(* CODESYS project UralKoksWin.project

Project tree, tasks and I/O mapping:
  Device : SPK1xx[M01], Production association OWEN, order no. 4, version 3.5.11.54
    application Application
      libraries: Standard, * (System); Util, * (System)
      task MainTask (cyclic, interval t#20ms, priority 1) calls PLC_PRG, MECH
      task VISU_TASK (cyclic, interval 100 ms, priority 31) calls VisuElems.Visu_Prg, CountWebCli
      task Task_Chain (cyclic, interval t#20ms, priority 1) calls Chain
      task TrendRecordingTask (cyclic, interval 100 ms, priority 31) calls VisuTrendStorageAccess.GlobalInstances.g_TrendRecordingManager.CyclicCall
      program PLC_PRG [LD]
      visualisation VFrADiag
      data type MV210_202
      data type MU210_402
      data type Vector75
      visualisation VMain
      visualisation VFr1Main
      image pool ImagePool
      visualisation VFr2Konv
      visualisation VFr3Grohot
      data type Vector100
      data type ABB330
      global variables GVL
      program MECH [CFC]
      data type PME
      program Chain [ST]
      function block Motor [LD]
      program CountWebCli [ST]
      visualisation VFr7RandE
    Info : Info, Production association OWEN, version 3.5.11.5002
        unmapped channels: VENDOR, DEVICE, SERIAL, RUNTIME, FIRMWARE, LINUX, TARGET, PROJECT, AUTHOR, VERSION, PROFILE, LASTCHANGES
    Screen : Screen, Production association OWEN, version 3.5.11.5001
        unmapped channels: Get Brightness, Dim time, Off time, Full brightness, Dim brightness, Off brightness, Dim visu name, Off visu name, On visu name, Wake up
    Debug : Debug, Production association OWEN, version 3.5.11.5001
        unmapped channels: RAM used, RAM free, Open files, Processor usage, Core temp, Enable Debug, Debug pause
    OwenRTC : OwenRTC, Production association OWEN, version 3.5.11.5001
        unmapped channels: Year, Month, Day, Hour, Minute, Second, Day of Week, Week of Year, Format Date, Format Time, UTC Offset, NTP Enabled, NTP Error, System Timer, New Year, New Month, New Day, New Hour, New Minute, New Second, New UTC Offset, Set Settings DT, Enable NTP, Prefer Server
    OwenCloud : OwenCloud, Production association OWEN, version 3.5.11.5001
        unmapped channels: OwenCloud enabled, Enable OwenCloud, Token
    Drives : Drives, Production association OWEN, version 3.5.11.5001
        unmapped channels: FS size, FS used, FS free, USB Mounted, USB Unmount done, USB size, USB used, USB free, MMC Mounted, MMC Unmount done, MMC size, MMC used, MMC free, Enable Drives, USB Unmount, MMC Unmount
    Network : Network, Production association OWEN, version 3.5.11.5001
        unmapped channels: DHCP enabled, IP, Mask, Gateway, MAC, Hostname, Enable DHCP, New IP, New Mask, New Gateway, New Hostname, Set Settings
    Watchdog : Watchdog, Production association OWEN, version 3.5.11.5001
        unmapped channels: Exception Handling, Last Exception Code, Last Exception Description, Last Exception Time, Hardware Watchdog Flag, Reboot
    Buzzer : Buzzer, Production association OWEN, version 3.5.11.5001
        unmapped channels: Buzzer enabled, Enable Buzzer
    Ethernet : Ethernet, 3S - Smart Software Solutions GmbH, version 3.5.11.0
        settings: IPAddress = [192,168,1,151]; SubnetMask = [255,255,255,0]; GatewayAddress = [0,0,0,0]; MACAddress = [16#E4,16#1E,16#0A,16#00,16#16,16#C1]; NetworkInterfaceName = 'eth0'; NetworkInterfaceName = "eth0"; SaveCommunicationSettings = FALSE
      Modbus_TCP_Master : Modbus TCP Master, 3S - Smart Software Solutions GmbH, version 3.5.11.30
          settings: AutoReconnect = TRUE
        MU210_402DO : Modbus TCP Slave, 3S - Smart Software Solutions GmbH, version 3.5.11.30
            settings: Unit-ID = 1; IPAddress = [192, 168, 1, 153]; DO.Function Code = 16; DO.Read Offset = 0; DO.Read Length = 0; DO.Write Offset = 16#01D6; DO.Write Length = 1; DO.Cycle Time = 20
            output Application.MECH.KMusor.xMODBUS_Run : BOOL  // DO.DO.Bit0
            output Application.MECH.KMagnit.xMODBUS_Run : BOOL  // DO.DO.Bit1
            output Application.MECH.K1.xMODBUS_Run : BOOL  // DO.DO.Bit2
            output Application.MECH.K3.xOUT_Run : BOOL  // DO.DO.Bit3
            output Application.MECH.Gr.xOUT_Run : BOOL  // DO.DO.Bit4
            output Application.MECH.K2.xMODBUS_Run : BOOL  // DO.DO.Bit5
            output Application.Chain.xLampPUSK : BOOL  // DO.DO.Bit13
            unmapped channels: DO
        MV210_202DI : Modbus TCP Slave, 3S - Smart Software Solutions GmbH, version 3.5.11.30
            settings: Unit-ID = 1; IPAddress = [192, 168, 1, 152]; DI.Function Code = 3; DI.Read Offset = 16#0033; DI.Read Length = 2; DI.Write Offset = 0; DI.Write Length = 0; DI.Cycle Time = 20
            input  Application.PLC_PRG.DInput1.xDI1 : BOOL  // DI.DI.Bit0
            input  Application.PLC_PRG.DInput1.xDI2 : BOOL  // DI.DI.Bit1
            input  Application.PLC_PRG.DInput1.xDI3 : BOOL  // DI.DI.Bit2
            input  Application.PLC_PRG.DInput1.xDI4 : BOOL  // DI.DI.Bit3
            input  Application.PLC_PRG.DInput1.xDI5 : BOOL  // DI.DI.Bit4
            input  Application.PLC_PRG.DInput1.xDI6 : BOOL  // DI.DI.Bit5
            input  Application.PLC_PRG.DInput1.xDI7 : BOOL  // DI.DI.Bit6
            input  Application.PLC_PRG.DInput1.xDI8 : BOOL  // DI.DI.Bit7
            input  Application.PLC_PRG.DInput1.xDI9 : BOOL  // DI.DI.Bit8
            input  Application.PLC_PRG.DInput1.xDI10 : BOOL  // DI.DI.Bit9
            input  Application.PLC_PRG.DInput1.xDI11 : BOOL  // DI.DI.Bit10
            input  Application.PLC_PRG.DInput1.xDI12 : BOOL  // DI.DI.Bit11
            input  Application.PLC_PRG.DInput1.xDI13 : BOOL  // DI.DI.Bit12
            input  Application.PLC_PRG.DInput1.xDI14 : BOOL  // DI.DI.Bit13
            input  Application.PLC_PRG.DInput1.xDI15 : BOOL  // DI.DI.Bit14
            input  Application.PLC_PRG.DInput1.xDI16 : BOOL  // DI.DI.Bit15
            input  Application.PLC_PRG.DInput1.xDI17 : BOOL  // DI.DI.Bit0
            input  Application.PLC_PRG.DInput1.xDI18 : BOOL  // DI.DI.Bit1
            input  Application.PLC_PRG.DInput1.xDI19 : BOOL  // DI.DI.Bit2
            input  Application.PLC_PRG.DInput1.xDI20 : BOOL  // DI.DI.Bit3
            unmapped channels: DI
        MV210_202DI2 : Modbus TCP Slave, 3S - Smart Software Solutions GmbH, version 3.5.11.30
            settings: Unit-ID = 1; IPAddress = [192, 168, 1, 154]; DI.Function Code = 3; DI.Read Offset = 16#0033; DI.Read Length = 2; DI.Write Offset = 0; DI.Write Length = 0; DI.Cycle Time = 20
            input  Application.PLC_PRG.DInput2.xDI1 : BOOL  // DI.DI.Bit0
            input  Application.PLC_PRG.DInput2.xDI2 : BOOL  // DI.DI.Bit1
            input  Application.PLC_PRG.DInput2.xDI6 : BOOL  // DI.DI.Bit5
            input  Application.PLC_PRG.DInput2.xDI7 : BOOL  // DI.DI.Bit6
            input  Application.PLC_PRG.DInput2.xDI8 : BOOL  // DI.DI.Bit7
            input  Application.PLC_PRG.DInput2.xDI9 : BOOL  // DI.DI.Bit8
            input  Application.PLC_PRG.DInput2.xDI10 : BOOL  // DI.DI.Bit9
            input  Application.PLC_PRG.DInput2.xDI11 : BOOL  // DI.DI.Bit10
            input  Application.PLC_PRG.DInput2.xDI12 : BOOL  // DI.DI.Bit11
            input  Application.PLC_PRG.DInput2.xDI13 : BOOL  // DI.DI.Bit12
            input  Application.PLC_PRG.DInput2.xDI14 : BOOL  // DI.DI.Bit13
            input  Application.PLC_PRG.DInput2.xDI15 : BOOL  // DI.DI.Bit14
            input  Application.PLC_PRG.DInput2.xDI16 : BOOL  // DI.DI.Bit15
            input  Application.PLC_PRG.DInput2.xDI17 : BOOL  // DI.DI.Bit0
            input  Application.PLC_PRG.DInput2.xDI18 : BOOL  // DI.DI.Bit1
            input  Application.PLC_PRG.DInput2.xDI19 : BOOL  // DI.DI.Bit2
            input  Application.PLC_PRG.DInput2.xDI20 : BOOL  // DI.DI.Bit3
            unmapped channels: DI
    COM1 : Modbus COM, 3S - Smart Software Solutions GmbH, version 3.5.11.20
        settings: DataBits = 8; StopBits = 2; ComPort = 1
      Master_1 : Modbus Master, COM Port, 3S - Smart Software Solutions GmbH, version 3.5.11.20
          settings: Transmission = 'RTU'; ResponseTimeout = 1000; TimeBetweenFrames = 10; Auto-restart communication = TRUE
        KonvMusorSlave : Modbus Slave, COM Port, 3S - Smart Software Solutions GmbH, version 3.5.10.30
            settings: SlaveAddress = 5; ResponseTimeout = 1000; UseExtendedFunctionCodes = TRUE; SPSpeed.Function Code = 6; SPSpeed.Read Offset = 0; SPSpeed.Read Length = 0; SPSpeed.Write Offset = 16#1000; SPSpeed.Write Length = 1; SPSpeed.Cycle Time = 1000; PVSpeed.Function Code = 3; PVSpeed.Read Offset = 16#1001; PVSpeed.Read Length = 1; PVSpeed.Write Offset = 0; PVSpeed.Write Length = 0; PVSpeed.Cycle Time = 1000; Current.Function Code = 3; Current.Read Offset = 16#1004; Current.Read Length = 1; Current.Write Offset = 0; Current.Write Length = 0; Current.Cycle Time = 1000; MI.Function Code = 3; MI.Read Offset = 16#1008; MI.Read Length = 1; MI.Write Offset = 0; MI.Write Length = 0; MI.Cycle Time = 1000
            output Application.MECH.KMusor.iMODBUS_SPSpeed : WORD  // SPSpeed.SPSpeed
            input  Application.MECH.KMusor.iMODBUS_PVSpeed : WORD  // PVSpeed.PVSpeed
            input  Application.MECH.KMusor.iMODBUS_Iengie : WORD  // Current.Current
            input  Application.MECH.KM_Konveer3 : BOOL  // MI.MI.Bit3
            input  Application.MECH.KM_Gr : BOOL  // MI.MI.Bit4
            unmapped channels: SPSpeed, PVSpeed, Current, MI
        Konv2Slave : Modbus Slave, COM Port, 3S - Smart Software Solutions GmbH, version 3.5.10.30
            settings: SlaveAddress = 20; ResponseTimeout = 1000; UseExtendedFunctionCodes = TRUE; PVSpeed.Function Code = 3; PVSpeed.Read Offset = 16#0004; PVSpeed.Read Length = 3; PVSpeed.Write Offset = 0; PVSpeed.Write Length = 0; PVSpeed.Cycle Time = 1000
            input  Application.MECH.K2.iMODBUS_SPSpeed : WORD  // PVSpeed.PVSpeed
            input  Application.MECH.K2.iMODBUS_PVSpeed : WORD  // PVSpeed.PVSpeed
            input  Application.MECH.K2.iMODBUS_Iengie : WORD  // PVSpeed.PVSpeed
            unmapped channels: PVSpeed
        KonvMagnitSlave : Modbus Slave, COM Port, 3S - Smart Software Solutions GmbH, version 3.5.10.30
            settings: SlaveAddress = 10; ResponseTimeout = 1000; UseExtendedFunctionCodes = TRUE; SPSpeed.Function Code = 6; SPSpeed.Read Offset = 0; SPSpeed.Read Length = 0; SPSpeed.Write Offset = 16#1000; SPSpeed.Write Length = 1; SPSpeed.Cycle Time = 1000; PVSpeed.Function Code = 3; PVSpeed.Read Offset = 16#1001; PVSpeed.Read Length = 1; PVSpeed.Write Offset = 0; PVSpeed.Write Length = 0; PVSpeed.Cycle Time = 1000; Current.Function Code = 3; Current.Read Offset = 16#1004; Current.Read Length = 1; Current.Write Offset = 0; Current.Write Length = 0; Current.Cycle Time = 1000
            output Application.MECH.KMagnit.iMODBUS_SPSpeed : WORD  // SPSpeed.SPSpeed
            input  Application.MECH.KMagnit.iMODBUS_PVSpeed : WORD  // PVSpeed.PVSpeed
            input  Application.MECH.KMagnit.iMODBUS_Iengie : WORD  // Current.Current
            unmapped channels: SPSpeed, PVSpeed, Current
        Konv1Slave : Modbus Slave, COM Port, 3S - Smart Software Solutions GmbH, version 3.5.10.30
            settings: SlaveAddress = 15; ResponseTimeout = 1000; UseExtendedFunctionCodes = TRUE; SPSpeed.Function Code = 6; SPSpeed.Read Offset = 0; SPSpeed.Read Length = 0; SPSpeed.Write Offset = 16#1000; SPSpeed.Write Length = 1; SPSpeed.Cycle Time = 1000; PVSpeed.Function Code = 3; PVSpeed.Read Offset = 16#1001; PVSpeed.Read Length = 1; PVSpeed.Write Offset = 0; PVSpeed.Write Length = 0; PVSpeed.Cycle Time = 1000; Current.Function Code = 3; Current.Read Offset = 16#1004; Current.Read Length = 1; Current.Write Offset = 0; Current.Write Length = 0; Current.Cycle Time = 1000
            output Application.MECH.K1.iMODBUS_SPSpeed : WORD  // SPSpeed.SPSpeed
            input  Application.MECH.K1.iMODBUS_PVSpeed : WORD  // PVSpeed.PVSpeed
            input  Application.MECH.K1.iMODBUS_Iengie : WORD  // Current.Current
            unmapped channels: SPSpeed, PVSpeed, Current
  text list GlobalTextList
  5ce3da45-db07-42e7-a21c-a00fff4ed8f6|img\fonFrame.png
  text list System
  5ce3da45-db07-42e7-a21c-a00fff4ed8f6|img\frame1.png
  5ce3da45-db07-42e7-a21c-a00fff4ed8f6|img\333.png
*)

// Device/Application/MV210_202
TYPE MV210_202 :
STRUCT
	xDI1: BOOL;
	xDI2: BOOL;
	xDI3: BOOL;
	xDI4: BOOL;
	xDI5: BOOL;
	xDI6: BOOL;
	xDI7: BOOL;
	xDI8: BOOL;
	xDI9: BOOL;
	xDI10: BOOL;
	xDI11: BOOL;
	xDI12: BOOL;
	xDI13: BOOL;
	xDI14: BOOL;
	xDI15: BOOL;
	xDI16: BOOL;
	xDI17: BOOL;
	xDI18: BOOL;
	xDI19: BOOL;
	xDI20: BOOL;
END_STRUCT
END_TYPE

// Device/Application/MU210_402
TYPE MU210_402 :
STRUCT
	xDO1: BOOL;
	xDO2: BOOL;
	xDO3: BOOL;
	xDO4: BOOL;
	xDO5: BOOL;
	xDO6: BOOL;
	xDO7: BOOL;
	xDO8: BOOL;
	xDO9: BOOL;
	xDO10: BOOL;
	xDO11: BOOL;
	xDO12: BOOL;
	xDO13: BOOL;
	xDO14: BOOL;
	xDO15: BOOL;
	xDO16: BOOL;
END_STRUCT
END_TYPE

// Device/Application/Vector75
TYPE Vector75 :
STRUCT
	iOUT_MODBUS_SPSpeed,
	iIN_MODBUS_PVSpeed,
	iIN_MODBUS_Iengie: INT;
	

	xIN_Run: BOOL;
	xOUT_MODBUS_Run:BOOL;
	xOUT_Ready: BOOL;
	xOUT_Error: BOOL;
	xOUT_Work: BOOL;

	xIN_Error: BOOL;

	iOUT_PVRotation: INT;
	iOUT_PVSpeed: INT; 

	rOUT_Current: REAL;
	
	iIN_MODBUS_AI: INT;
END_STRUCT
END_TYPE

// Device/Application/Vector100
TYPE Vector100 :
STRUCT
	iMODBUS_SPSpeed,
	iMODBUS_PVSpeed,
	iMODBUS_Iengie: INT;
	

	xIN_Run: BOOL;
	xMODBUS_Run:BOOL;
	xOUT_Ready: BOOL;
	xOUT_Error: BOOL;
	xOUT_Work: BOOL;

	xIN_Error: BOOL;

	iOUT_PVRotation: INT;
	iOUT_PVSpeed: INT; 

	rOUT_Current: REAL;
	
END_STRUCT
END_TYPE

// Device/Application/ABB330
TYPE ABB330 :
STRUCT
	iMODBUS_SPSpeed,
	iMODBUS_PVSpeed,
	iMODBUS_Iengie: INT;
	

	xIN_Run: BOOL;
	xMODBUS_Run:BOOL;
	xOUT_Ready: BOOL;
	xOUT_Error: BOOL;
	xOUT_Work: BOOL;

	xIN_Error: BOOL;

	iOUT_PVRotation: INT;
	iOUT_PVSpeed: INT; 

	rOUT_Current: REAL;
	
END_STRUCT
END_TYPE

// Device/Application/PME
TYPE PME :
STRUCT

	xIN_Run: BOOL;
	xIN_Error: BOOL;

	
	
	xOUT_Ready: BOOL;
	xOUT_Error: BOOL;
	xOUT_Work: BOOL;
	xOUT_Run: BOOL;
	
	iOUT_PVSpeed: INT;
	

	iOUT_PVRotation: INT;
	
END_STRUCT
END_TYPE

// Device/Application/GVL
{attribute 'qualified_only'}
VAR_GLOBAL

END_VAR

// Device/Application/PLC_PRG
PROGRAM PLC_PRG
VAR

	xAck :BOOL;
	DInput1: MV210_202;
	DInput2: MV210_202;
	DOutput1: MU210_402;
	xFlash: BOOL;
	Flasing: BLINK;
	Sechka: SR;
	Drob: SR;
END_VAR

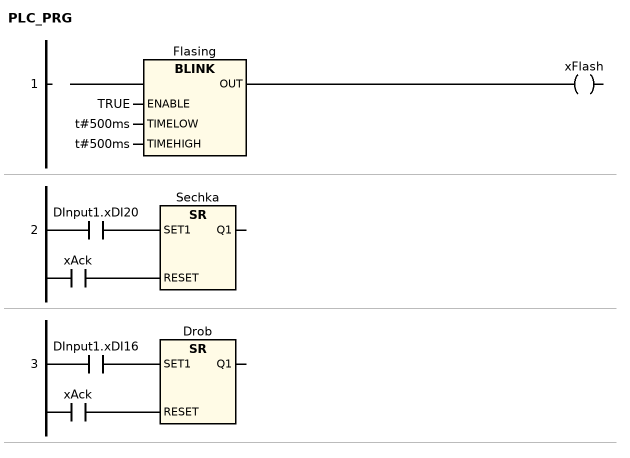
// NETWORK 1
Flasing(ENABLE := TRUE, TIMELOW := t#500ms, TIMEHIGH := t#500ms); // BLINK
xFlash := Flasing.OUT;

// NETWORK 2
Sechka(SET1 := DInput1.xDI20, RESET := xAck); // SR

// NETWORK 3
Drob(SET1 := DInput1.xDI16, RESET := xAck); // SR

END_PROGRAM

// Device/Application/MECH
PROGRAM MECH
VAR
	KonveerMusor: Motor;
	KonveerMagnit: Motor;
	Konveer1: Motor;
	Konveer3: Motor;
	Grohot: Motor;
	Konveer2: Motor;


	iSP_Konveer2: INT;

	KM_Konveer3: BOOL;
	KM_Gr: BOOL;
END_VAR

VAR_INPUT
	KMusor:Vector100;
	KMagnit:Vector100;
	K1:Vector100;
	K3: PME;
	Gr: PME;
	K2: ABB330;
END_VAR

VAR RETAIN
	KMusor_iIN_SPSpeed: INT:=20;
	KMusor_xIN_EnCtrlSensor: BOOL:=TRUE;
	KMusor_iIN_SPRotatTimeMS: INT:=6300;
	
	KMagnit_iIN_SPSpeed: INT:=25;

	
	K1_xIN_EnCtrlSensor: BOOL:=TRUE;
	K1_iIN_SPSpeed: INT:=30;
	K1_iIN_SPRotatTimeMS: INT:=3000;
	
	K3_xIN_EnCtrlSensor: BOOL:=TRUE;
	K3_iIN_SPRotatTimeMS: INT:=3000;
	
	K2_iIN_SPSpeed: INT:=27;
	K2_xIN_EnCtrlSensor: BOOL:=TRUE;
	K2_iIN_SPRotatTimeMS: INT:=3000;	
END_VAR
VAR // added by the converter: edge detectors and wires of the graphical bodies
    _w1 : ANY;
    _w2 : INT;
END_VAR

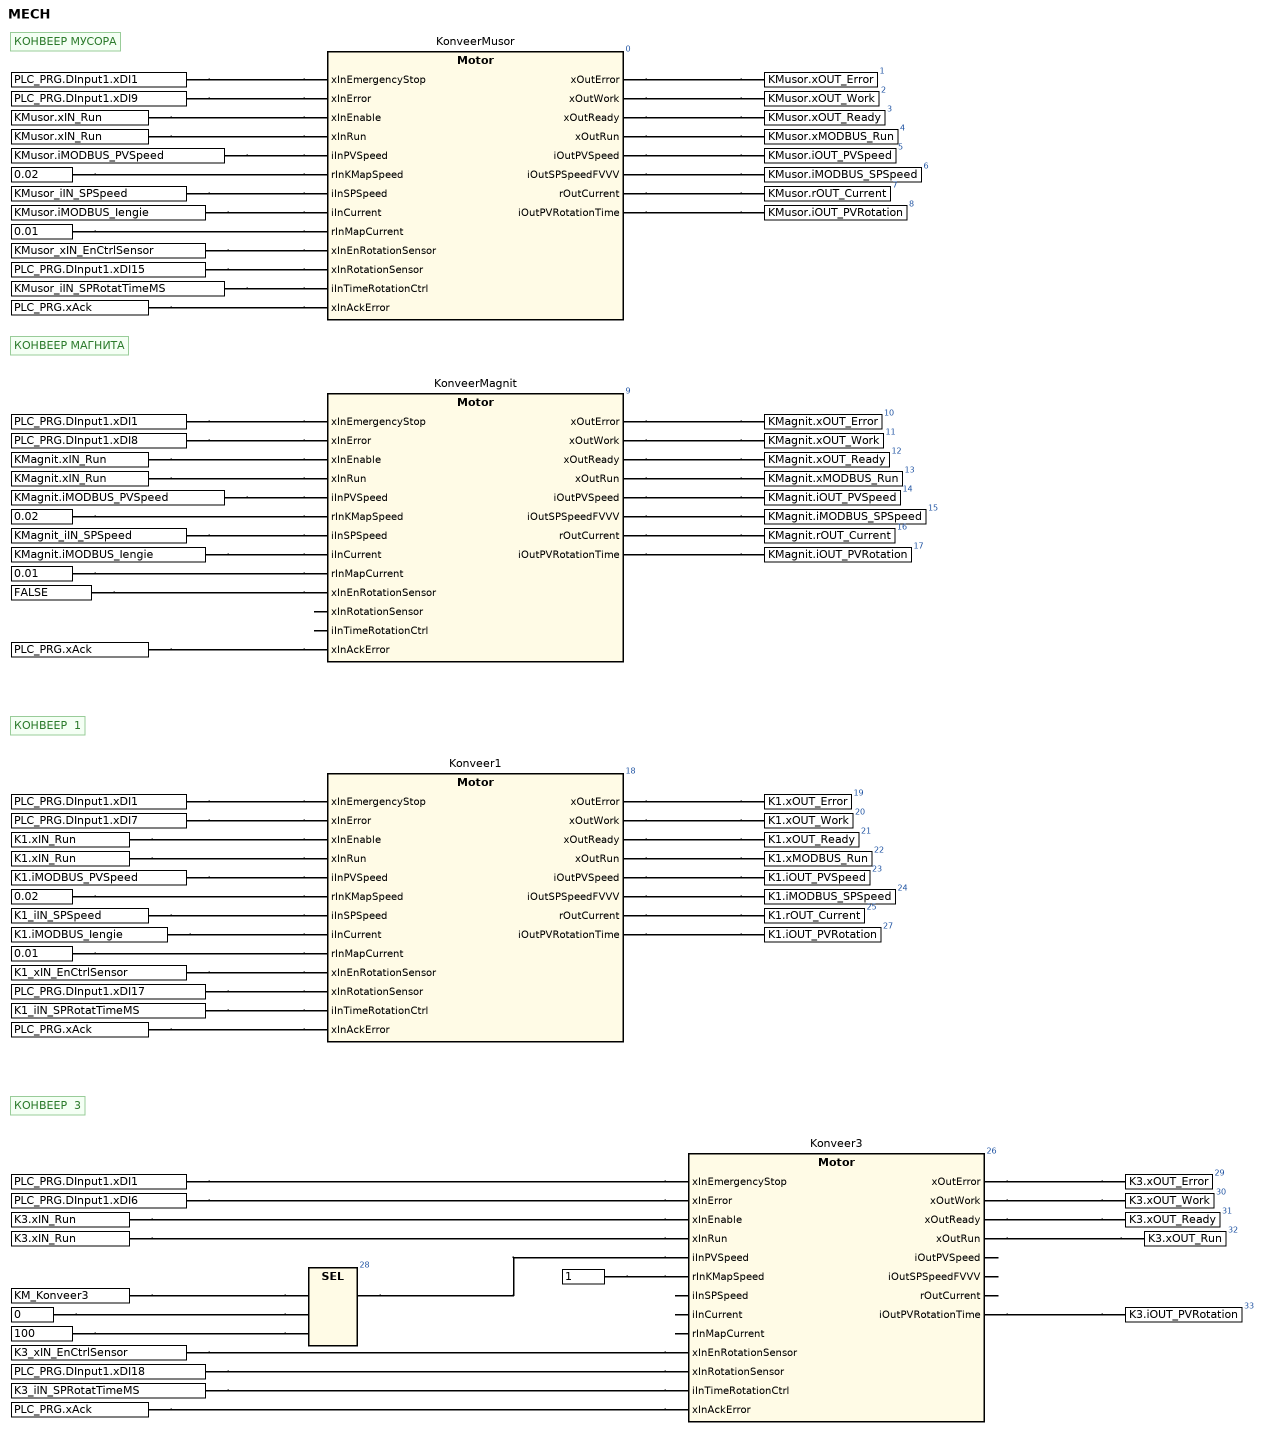
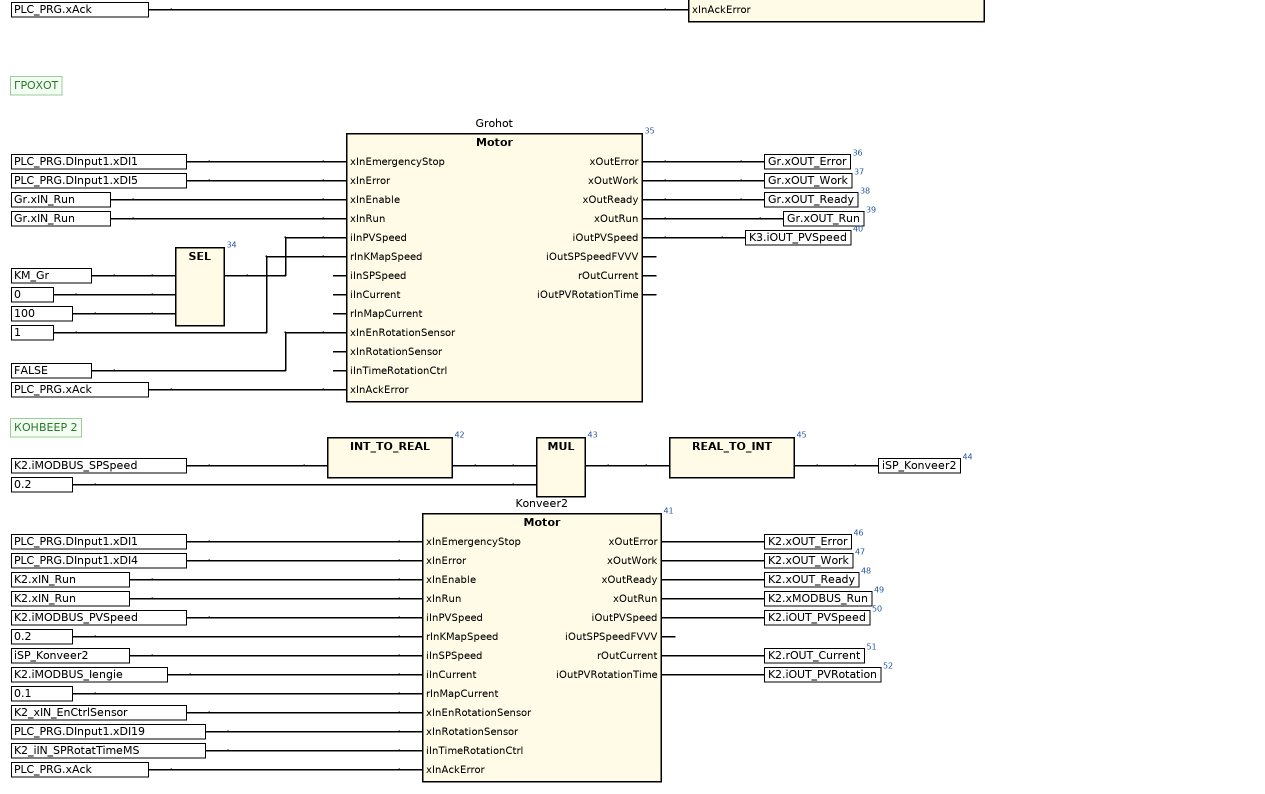
// note: 117 stored wires end on pins the file does not list and are not shown
// КОНВЕЕР МУСОРА
KonveerMusor(
    xInEmergencyStop := PLC_PRG.DInput1.xDI1,
    xInError := PLC_PRG.DInput1.xDI9,
    xInEnable := KMusor.xIN_Run,
    xInRun := KMusor.xIN_Run,
    iInPVSpeed := KMusor.iMODBUS_PVSpeed,
    rInKMapSpeed := 0.02,
    iInSPSpeed := KMusor_iIN_SPSpeed,
    iInCurrent := KMusor.iMODBUS_Iengie,
    rInMapCurrent := 0.01,
    xInEnRotationSensor := KMusor_xIN_EnCtrlSensor,
    xInRotationSensor := PLC_PRG.DInput1.xDI15,
    iInTimeRotationCtrl := KMusor_iIN_SPRotatTimeMS,
    xInAckError := PLC_PRG.xAck); // Motor
KMusor.xOUT_Error := KonveerMusor.xOutError;
KMusor.xOUT_Work := KonveerMusor.xOutWork;
KMusor.xOUT_Ready := KonveerMusor.xOutReady;
KMusor.xMODBUS_Run := KonveerMusor.xOutRun;
KMusor.iOUT_PVSpeed := KonveerMusor.iOutPVSpeed;
KMusor.iMODBUS_SPSpeed := KonveerMusor.iOutSPSpeedFVVV;
KMusor.rOUT_Current := KonveerMusor.rOutCurrent;
KMusor.iOUT_PVRotation := KonveerMusor.iOutPVRotationTime;
// КОНВЕЕР МАГНИТА
KonveerMagnit(
    xInEmergencyStop := PLC_PRG.DInput1.xDI1,
    xInError := PLC_PRG.DInput1.xDI8,
    xInEnable := KMagnit.xIN_Run,
    xInRun := KMagnit.xIN_Run,
    iInPVSpeed := KMagnit.iMODBUS_PVSpeed,
    rInKMapSpeed := 0.02,
    iInSPSpeed := KMagnit_iIN_SPSpeed,
    iInCurrent := KMagnit.iMODBUS_Iengie,
    rInMapCurrent := 0.01,
    xInEnRotationSensor := FALSE,
    xInAckError := PLC_PRG.xAck); // Motor
KMagnit.xOUT_Error := KonveerMagnit.xOutError;
KMagnit.xOUT_Work := KonveerMagnit.xOutWork;
KMagnit.xOUT_Ready := KonveerMagnit.xOutReady;
KMagnit.xMODBUS_Run := KonveerMagnit.xOutRun;
KMagnit.iOUT_PVSpeed := KonveerMagnit.iOutPVSpeed;
KMagnit.iMODBUS_SPSpeed := KonveerMagnit.iOutSPSpeedFVVV;
KMagnit.rOUT_Current := KonveerMagnit.rOutCurrent;
KMagnit.iOUT_PVRotation := KonveerMagnit.iOutPVRotationTime;
// КОНВЕЕР  1
Konveer1(
    xInEmergencyStop := PLC_PRG.DInput1.xDI1,
    xInError := PLC_PRG.DInput1.xDI7,
    xInEnable := K1.xIN_Run,
    xInRun := K1.xIN_Run,
    iInPVSpeed := K1.iMODBUS_PVSpeed,
    rInKMapSpeed := 0.02,
    iInSPSpeed := K1_iIN_SPSpeed,
    iInCurrent := K1.iMODBUS_Iengie,
    rInMapCurrent := 0.01,
    xInEnRotationSensor := K1_xIN_EnCtrlSensor,
    xInRotationSensor := PLC_PRG.DInput1.xDI17,
    iInTimeRotationCtrl := K1_iIN_SPRotatTimeMS,
    xInAckError := PLC_PRG.xAck); // Motor
K1.xOUT_Error := Konveer1.xOutError;
K1.xOUT_Work := Konveer1.xOutWork;
K1.xOUT_Ready := Konveer1.xOutReady;
K1.xMODBUS_Run := Konveer1.xOutRun;
K1.iOUT_PVSpeed := Konveer1.iOutPVSpeed;
K1.iMODBUS_SPSpeed := Konveer1.iOutSPSpeedFVVV;
K1.rOUT_Current := Konveer1.rOutCurrent;
Konveer3(
    xInEmergencyStop := PLC_PRG.DInput1.xDI1,
    xInError := PLC_PRG.DInput1.xDI6,
    xInEnable := K3.xIN_Run,
    xInRun := K3.xIN_Run,
    iInPVSpeed := _w1,
    rInKMapSpeed := 1,
    xInEnRotationSensor := K3_xIN_EnCtrlSensor,
    xInRotationSensor := PLC_PRG.DInput1.xDI18,
    iInTimeRotationCtrl := K3_iIN_SPRotatTimeMS,
    xInAckError := PLC_PRG.xAck); // Motor
K1.iOUT_PVRotation := Konveer1.iOutPVRotationTime;
// КОНВЕЕР  3
_w1 := SEL(KM_Konveer3, 0, 100);
K3.xOUT_Error := Konveer3.xOutError;
K3.xOUT_Work := Konveer3.xOutWork;
K3.xOUT_Ready := Konveer3.xOutReady;
K3.xOUT_Run := Konveer3.xOutRun;
K3.iOUT_PVRotation := Konveer3.iOutPVRotationTime;
// ГРОХОТ
Grohot(
    xInEmergencyStop := PLC_PRG.DInput1.xDI1,
    xInError := PLC_PRG.DInput1.xDI5,
    xInEnable := Gr.xIN_Run,
    xInRun := Gr.xIN_Run,
    iInPVSpeed := SEL(KM_Gr, 0, 100),
    rInKMapSpeed := 1,
    xInEnRotationSensor := FALSE,
    xInAckError := PLC_PRG.xAck); // Motor
Gr.xOUT_Error := Grohot.xOutError;
Gr.xOUT_Work := Grohot.xOutWork;
Gr.xOUT_Ready := Grohot.xOutReady;
Gr.xOUT_Run := Grohot.xOutRun;
K3.iOUT_PVSpeed := Grohot.iOutPVSpeed;
Konveer2(
    xInEmergencyStop := PLC_PRG.DInput1.xDI1,
    xInError := PLC_PRG.DInput1.xDI4,
    xInEnable := K2.xIN_Run,
    xInRun := K2.xIN_Run,
    iInPVSpeed := K2.iMODBUS_PVSpeed,
    rInKMapSpeed := 0.2,
    iInSPSpeed := iSP_Konveer2,
    iInCurrent := K2.iMODBUS_Iengie,
    rInMapCurrent := 0.1,
    xInEnRotationSensor := K2_xIN_EnCtrlSensor,
    xInRotationSensor := PLC_PRG.DInput1.xDI19,
    iInTimeRotationCtrl := K2_iIN_SPRotatTimeMS,
    xInAckError := PLC_PRG.xAck); // Motor
// КОНВЕЕР 2
iSP_Konveer2 := _w2;
_w2 := REAL_TO_INT(INT_TO_REAL(K2.iMODBUS_SPSpeed) * 0.2);
K2.xOUT_Error := Konveer2.xOutError;
K2.xOUT_Work := Konveer2.xOutWork;
K2.xOUT_Ready := Konveer2.xOutReady;
K2.xMODBUS_Run := Konveer2.xOutRun;
K2.iOUT_PVSpeed := Konveer2.iOutPVSpeed;
K2.rOUT_Current := Konveer2.rOutCurrent;
K2.iOUT_PVRotation := Konveer2.iOutPVRotationTime;

END_PROGRAM

// Device/Application/Motor
FUNCTION_BLOCK Motor
VAR_INPUT
	//Аварийный стоп
	xInEmergencyStop: BOOL;
	// Ошибка преобразователя
	xInError: BOOL;
	// Режим Использования
	xInEnable: BOOL;
	// Пуск
	xInRun: BOOL;
	
	//факт обороты
	iInPVSpeed: INT;
	//Коэф.маштабирования оборотов
	rInKMapSpeed: REAL;
	//Задание оборотов (0-100%)
	iInSPSpeed: INT;
	
	// Ток двигателя
	iInCurrent: INT;
	// Коэф маштабирования тока
	rInMapCurrent: REAL;
	
	// Контроль вращения Включить
	xInEnRotationSensor: BOOL;
	// Датчик контроля вращения
	xInRotationSensor: BOOL;
	// Время контороля вращения
	iInTimeRotationCtrl: INT;
	
	// Вход Подтвердить ошибку
	xInAckError: BOOL;
END_VAR
VAR_OUTPUT
	// Ошибка
	xOutError: BOOL;
	// Двигатель работает
	xOutWork: BOOL;
	//Готовность
	xOutReady: BOOL;
	// Команда ПУСК
	xOutRun: BOOL;
	

	//Факт частота вращения(0-100%)
	iOutPVSpeed: INT;
	// Задание частоты вращения(0-10000) для ПЧ
	iOutSPSpeedFVVV:INT;
	
	// Ток двигателя
	rOutCurrent: REAL;
	
	//Факт время оборота, мс
	iOutPVRotationTime: INT;
END_VAR

VAR
	// Готовность
	xReady: BOOL;
	// Команда Пуск
	xRun: BOOL;
	// Работает
	xWork1: BOOL;
	// Фактическое время вращения
	PVRotationTimeMilliSecund: TIME;
	// Заданное время вращения
	SPRotationTimeMilliSecund: TIME;

	xPFront: BOOL;
	xNFront: BOOL;
	T2: TON;
	T1: TON;
	xC: BOOL;
	rTemp1: REAL;
	rTemp2: REAL;
	xTemp1: BOOL;
	xFirstRun: BOOL;
	T0: TON;
	SPRotationTimeMilliSecund3: TIME;
	PVRotationTimeMilliSecund3: TIME;
	xStartNoRotation: BOOL;
	xNoRation: BOOL;
	xExtError: BOOL;
END_VAR
VAR // added by the converter: edge detectors and wires of the graphical bodies
    _rt1, _rt2, _rt3 : R_TRIG;
    _ft1, _ft2, _ft3 : F_TRIG;
    _w1, _w2 : BOOL;
END_VAR

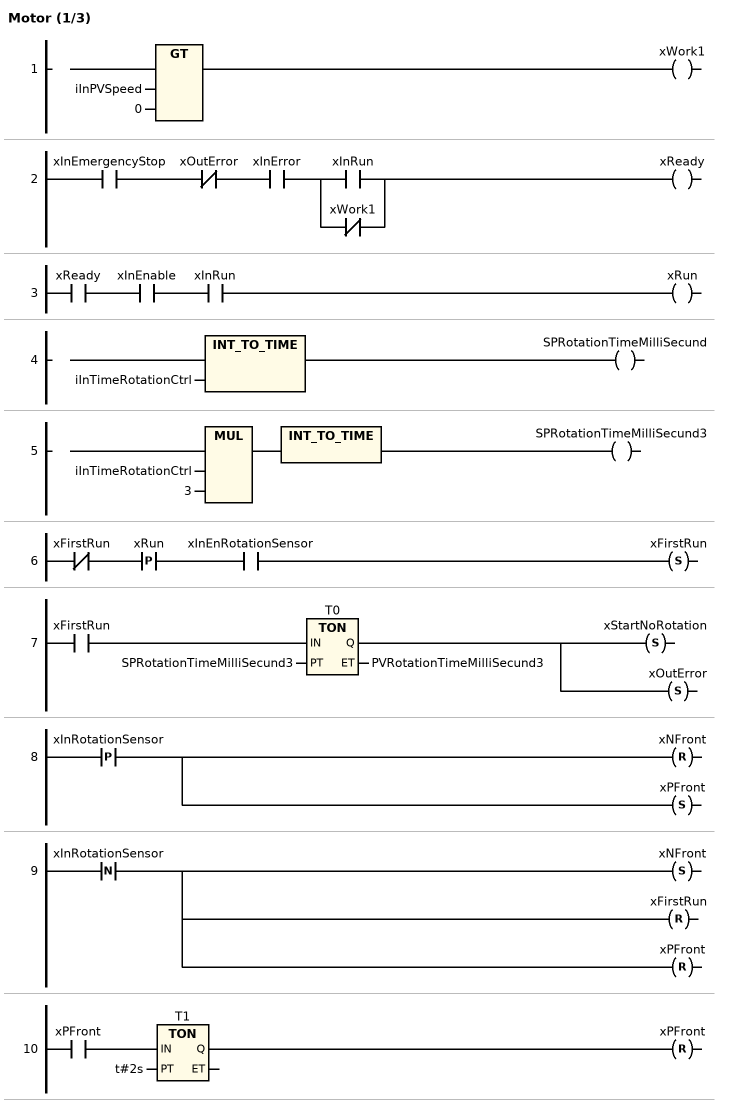
// NETWORK 1
xWork1 := iInPVSpeed > 0;

// NETWORK 2
xReady := xInEmergencyStop AND NOT xOutError AND xInError AND (xInRun OR NOT xWork1);

// NETWORK 3
xRun := xReady AND xInEnable AND xInRun;

// NETWORK 4
SPRotationTimeMilliSecund := INT_TO_TIME(iInTimeRotationCtrl);

// NETWORK 5
SPRotationTimeMilliSecund3 := INT_TO_TIME(iInTimeRotationCtrl * 3);

// NETWORK 6
_rt1(CLK := xRun);
xFirstRun S= NOT xFirstRun AND _rt1.Q AND xInEnRotationSensor;

// NETWORK 7
T0(IN := xFirstRun, PT := SPRotationTimeMilliSecund3, ET => PVRotationTimeMilliSecund3); // TON
xStartNoRotation S= T0.Q;
xOutError S= T0.Q;

// NETWORK 8
_rt2(CLK := xInRotationSensor);
xNFront R= _rt2.Q;
xPFront S= _rt2.Q;

// NETWORK 9
_ft1(CLK := xInRotationSensor);
xNFront S= _ft1.Q;
xFirstRun R= _ft1.Q;
xPFront R= _ft1.Q;

// NETWORK 10
T1(IN := xPFront, PT := t#2s); // TON
xPFront R= T1.Q;

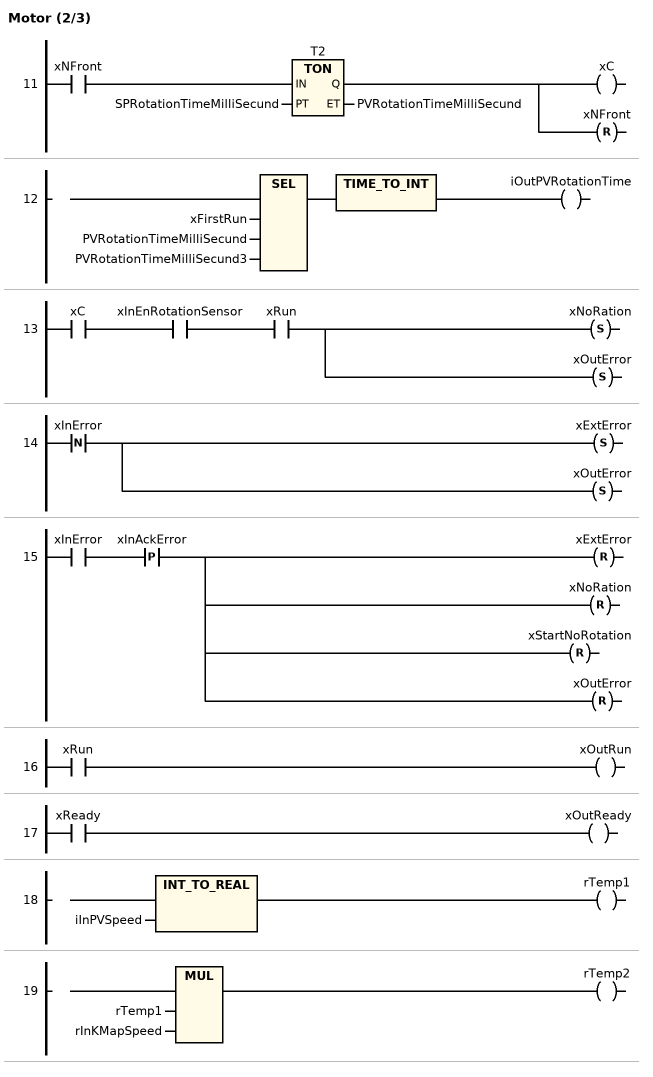
// NETWORK 11
T2(IN := xNFront, PT := SPRotationTimeMilliSecund, ET => PVRotationTimeMilliSecund); // TON
xC := T2.Q;
xNFront R= T2.Q;

// NETWORK 12
iOutPVRotationTime := TIME_TO_INT(SEL(xFirstRun, PVRotationTimeMilliSecund, PVRotationTimeMilliSecund3));

// NETWORK 13
_w1 := xC AND xInEnRotationSensor AND xRun;
xNoRation S= _w1;
xOutError S= _w1;

// NETWORK 14
_ft2(CLK := xInError);
xExtError S= _ft2.Q;
xOutError S= _ft2.Q;

// NETWORK 15
_rt3(CLK := xInAckError);
_w2 := xInError AND _rt3.Q;
xExtError R= _w2;
xNoRation R= _w2;
xStartNoRotation R= _w2;
xOutError R= _w2;

// NETWORK 16
xOutRun := xRun;

// NETWORK 17
xOutReady := xReady;

// NETWORK 18
rTemp1 := INT_TO_REAL(iInPVSpeed);

// NETWORK 19
rTemp2 := rTemp1 * rInKMapSpeed;

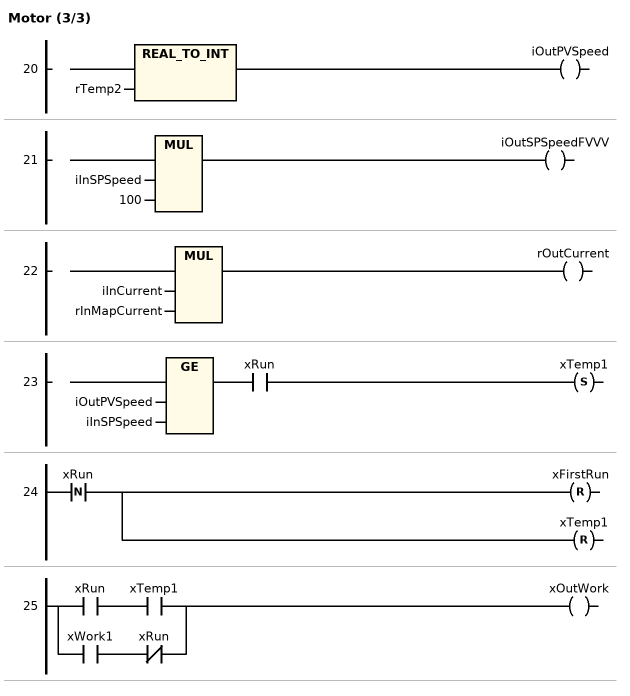
// NETWORK 20
iOutPVSpeed := REAL_TO_INT(rTemp2);

// NETWORK 21
iOutSPSpeedFVVV := iInSPSpeed * 100;

// NETWORK 22
rOutCurrent := iInCurrent * rInMapCurrent;

// NETWORK 23
xTemp1 S= iOutPVSpeed >= iInSPSpeed AND xRun;

// NETWORK 24
_ft3(CLK := xRun);
xFirstRun R= _ft3.Q;
xTemp1 R= _ft3.Q;

// NETWORK 25
xOutWork := xRun AND xTemp1 OR xWork1 AND NOT xRun;

END_FUNCTION_BLOCK

// Device/Application/CountWebCli
PROGRAM CountWebCli
VAR
	pClient: POINTER TO VisuElems.VisuStructClientData;
	iCountActivWebVisus: INT;
	xAlarm: BOOL;
END_VAR

iCountActivWebVisus:=0;
xAlarm:=FALSE;

VisuElems.VisuElemBase.g_ClientManager.BeginIteration();

WHILE (pClient:=VisuElems.VisuElemBase.g_ClientManager.GetNextClient())<>0 DO
	IF pClient^.GlobalData.ClientType = VisuElems.Visu_ClientType.Webvisualization THEN
		iCountActivWebVisus:=iCountActivWebVisus+1;
		xAlarm:=TRUE;
	END_IF
END_WHILE

END_PROGRAM

// Device/Application/Chain
PROGRAM Chain
VAR
	ReadyRun: BOOL:=FALSE;
	Run: BOOL:=FALSE;
	EmerSTOP: BOOL;
	Stop5: BOOL;	

	Step: INT:=0;

	TMR990: TON;
	Stoped995: BOOL;
	Runed5: BOOL;
	Stop10: BOOL;
	Runed10: BOOL;
	Stop: BOOL;
	Stoped990: BOOL;
	TMR5: TON;
	Stop15: BOOL;
	Runed15: BOOL;
	Stoped985: BOOL;
	Stop20: BOOL;
	Runed20: BOOL;
	TMR980: TON;
	Stop25: BOOL;
	Runed25: BOOL;
	TMR975: TON;
	Stop30: BOOL;
	TMRWork: TON;
	TMR970: TON;
	xLampPUSK: BOOL;
END_VAR

//IF <condition> THEN
//    <statements>
//( ELSIF <condition> THEN
//        <statements> )*
//( ELSE
//        <statements> )?
//END_IF;
// ( ... )* None, once or several times
// ( ... )? Optional

//	TMR995 (IN:=Step=995 AND NOT(TMR995.Q), PT:=T#5S);
//	IF TMR995.Q THEN
//		Step:=0;
//	END_IF

EmerSTOP:= NOT(PLC_PRG.DInput1.xDI1);

ReadyRun:= PLC_PRG.DInput1.xDI1 // ававрийный стоп
			AND MECH.KMusor.xOUT_Ready
			//AND MECH.KMagnit.xOUT_Ready
			AND MECH.K1.xOUT_Ready
			//AND MECH.K3.xOUT_Ready
			AND MECH.Gr.xOUT_Ready
			AND MECH.K2.xOUT_Ready
			AND NOT PLC_PRG.Sechka.Q1  //уровень дроби 1
			AND NOT PLC_PRG.Drob.Q1; //уровень дроби 2

			
Stop:=NOT(PLC_PRG.DInput1.xDI14);

			
Run:= PLC_PRG.DInput1.xDI13 
		AND PLC_PRG.DInput1.xDI14;

	
Runed5:= MECH.KMusor.xOUT_Work
		//AND MECH.KMagnit.xOUT_Work
		//AND MECH.K3.xOUT_Work
		AND MECH.Gr.xOUT_Work;

Runed10:= MECH.Gr.xOUT_Work;

Runed15:= MECH.K2.xOUT_Work;

Stop5:=   MECH.KMusor.xOUT_Error
		//OR MECH.KMagnit.xOUT_Error
		//OR MECH.K3.xOUT_Error
		OR MECH.Gr.xOUT_Error
		OR PLC_PRG.Sechka.Q1  //уровень дроби 1
		OR PLC_PRG.Drob.Q1; //уровень дроби 2
		
Stop10:= MECH.K1.xOUT_Error
		 OR MECH.K2.xOUT_Error;
		
Stoped995:=NOT(MECH.KMusor.xOUT_Work)
		//AND NOT(MECH.KMagnit.xOUT_Work)
		AND NOT(MECH.K1.xOUT_Work)
		//AND NOT(MECH.K3.xOUT_Work)
		AND NOT(MECH.Gr.xOUT_Work)
		AND NOT(MECH.K2.xOUT_Work);	


///===============================================================================================================================

IF Step=0 THEN
	IF ReadyRun THEN
		IF Run THEN
			Step:=5;
		END_IF;
		ELSE 
		Step:=1;
	END_IF;
ELSIF Step=1 THEN
	IF ReadyRun THEN
		Step:=0;
	END_IF

// ЗАПУСК КОНВЕЙЕРа 3, Мусора, Магнита, Грохота	
ELSIF Step=5 THEN
	MECH.KMusor.xIN_Run:=TRUE;
	//MECH.KMagnit.xIN_Run:=TRUE;
	//MECH.K3.xIN_Run:=TRUE;
	MECH.Gr.xIN_Run:=TRUE;
	xLampPUSK:=TRUE;
	IF Stop5 OR Stop THEN
		Step:=995;	
	END_IF;
	IF EmerSTOP THEN
		Step:=1000;
	END_IF;
	
	TMR5 (IN:=Step=5 AND NOT(TMR5.Q), PT:=T#10S);
	IF Runed5 AND TMR5.Q THEN
		Step:=10;		
	END_IF;

// ЗАПУСК Конвееров 1,2	
ELSIF Step=10 THEN	
	MECH.K1.xIN_Run:=TRUE;
	MECH.K2.xIN_Run:=TRUE;
	IF Stop5 OR Stop10 OR Stop THEN
		Step:=995;	
	END_IF;
	IF EmerSTOP THEN
		Step:=1000;
	END_IF;
		
//////////////=========================================

// ОСТАНОВКА
ELSIF Step=995 THEN
	MECH.KMusor.xIN_Run:=FALSE;
	//MECH.KMagnit.xIN_Run:=FALSE;
	MECH.K1.xIN_Run:=FALSE;
	//MECH.K3.xIN_Run:=FALSE;
	MECH.Gr.xIN_Run:=FALSE;
	MECH.K2.xIN_Run:=FALSE;
	xLampPUSK:=FALSE;
	IF Stoped995 THEN
		Step:=0;
	END_IF

// АВАРИЙНЫЙ СТОП!!	
ELSIF Step=1000 THEN
	MECH.KMusor.xIN_Run:=FALSE;
	//MECH.KMagnit.xIN_Run:=FALSE;
	MECH.K1.xIN_Run:=FALSE;
	//MECH.K3.xIN_Run:=FALSE;
	MECH.Gr.xIN_Run:=FALSE;
	MECH.K2.xIN_Run:=FALSE;
	xLampPUSK:=FALSE;
	IF	PLC_PRG.xAck AND Stoped995 THEN
		Step:=0;
	END_IF		
END_IF

END_PROGRAM

// Device/Application/VFrADiag
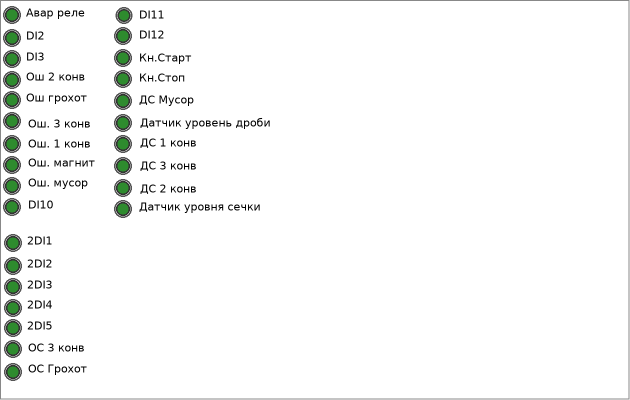
VISUALIZATION VFrADiag  // 630x400, background image ImagePool.fonFreame
    Lamp1 (2,5 20x20), variable: PLC_PRG.DInput1.xDI1, style: Lamp-Lamp1-Green
    Lamp1 (2,28 20x20), variable: PLC_PRG.DInput1.xDI2, style: Lamp-Lamp1-Green
    Lamp1 (2,49 20x20), variable: PLC_PRG.DInput1.xDI3, style: Lamp-Lamp1-Green
    Lamp1 (2,70 20x20), variable: PLC_PRG.DInput1.xDI4, style: Lamp-Lamp1-Green
    Lamp1 (2,90 20x20), variable: PLC_PRG.DInput1.xDI5, style: Lamp-Lamp1-Green
    Lamp1 (2,111 20x20), variable: PLC_PRG.DInput1.xDI6, style: Lamp-Lamp1-Green
    Lamp1 (2,134 20x20), variable: PLC_PRG.DInput1.xDI7, style: Lamp-Lamp1-Green
    Lamp1 (2,155 20x20), variable: PLC_PRG.DInput1.xDI8, style: Lamp-Lamp1-Green
    Lamp1 (2,176 20x20), variable: PLC_PRG.DInput1.xDI9, style: Lamp-Lamp1-Green
    Lamp1 (2,197 20x20), variable: PLC_PRG.DInput1.xDI10, style: Lamp-Lamp1-Green
    Lamp1 (113,6 22x19), variable: PLC_PRG.DInput1.xDI11, style: Lamp-Lamp1-Green
    Lamp1 (113,26 20x20), variable: PLC_PRG.DInput1.xDI12, style: Lamp-Lamp1-Green
    Lamp1 (113,48 20x20), variable: PLC_PRG.DInput1.xDI13, style: Lamp-Lamp1-Green
    Lamp1 (113,69 20x20), variable: PLC_PRG.DInput1.xDI14, style: Lamp-Lamp1-Green
    Lamp1 (113,91 20x20), variable: PLC_PRG.DInput1.xDI15, style: Lamp-Lamp1-Green
    Lamp1 (113,113 20x20), variable: PLC_PRG.DInput1.xDI16, style: Lamp-Lamp1-Green
    Lamp1 (113,134 20x20), variable: PLC_PRG.DInput1.xDI17, style: Lamp-Lamp1-Green
    Lamp1 (113,156 20x20), variable: PLC_PRG.DInput1.xDI18, style: Lamp-Lamp1-Green
    Lamp1 (113,178 20x20), variable: PLC_PRG.DInput1.xDI19, style: Lamp-Lamp1-Green
    Lamp1 (113,199 20x20), variable: PLC_PRG.DInput1.xDI20, style: Lamp-Lamp1-Green
    Label (23,-2 66x30), "Авар реле"
    Label (23,62 86x30), "Ош 2 конв"
    Label (23,83 83x30), "Ош грохот"
    Label (25,148 61x30), "Ош. магнит"
    Label (25,168 62x30), "Ош. мусор"
    Label (25,109 63x30), "Ош. 3 конв"
    Label (136,20 79x30), "DI12"
    Label (136,43 67x30), "Кн.Старт"
    Label (136,63 67x30), "Кн.Стоп"
    Label (136,85 83x30), "ДС Мусор"
    Label (25,190 34x30), "DI10"
    Label (136,0 53x30), "DI11"
    Label (23,21 93x30), "DI2"
    Label (23,42 89x30), "DI3"
    Label (25,129 63x30), "Ош. 1 конв"
    Label (137,108 139x30), "Датчик уровень дроби"
    Label (137,128 57x30), "ДС 1 конв"
    Label (137,151 84x30), "ДС 3 конв"
    Label (137,174 90x30), "ДС 2 конв"
    Label (136,192 130x30), "Датчик уровня сечки"
    Lamp1 (3,233 20x20), variable: PLC_PRG.DInput2.xDI1, style: Lamp-Lamp1-Green
    Lamp1 (3,256 20x20), variable: PLC_PRG.DInput2.xDI2, style: Lamp-Lamp1-Green
    Lamp1 (3,277 20x20), variable: PLC_PRG.DInput2.xDI3, style: Lamp-Lamp1-Green
    Lamp1 (3,298 20x20), variable: PLC_PRG.DInput2.xDI4, style: Lamp-Lamp1-Green
    Lamp1 (3,318 20x20), variable: PLC_PRG.DInput2.xDI5, style: Lamp-Lamp1-Green
    Lamp1 (3,339 20x20), variable: PLC_PRG.DInput2.xDI6, style: Lamp-Lamp1-Green
    Lamp1 (3,362 20x20), variable: PLC_PRG.DInput2.xDI7, style: Lamp-Lamp1-Green
    Label (24,226 66x30), "2DI1"
    Label (24,290 86x30), "2DI4"
    Label (24,311 83x30), "2DI5"
    Label (24,249 93x30), "2DI2"
    Label (24,270 89x30), "2DI3"
    Label (25,354 83x30), "ОС Грохот"
    Label (25,333 86x30), "ОС 3 конв"
END_VISUALIZATION

// Device/Application/VMain
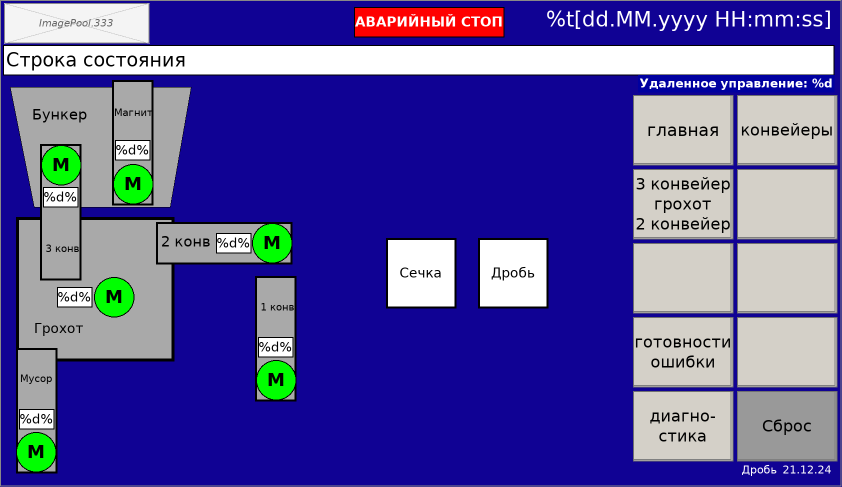
VISUALIZATION VMain  // 842x487
    Frame (-1,79 630x400)
        shows VFr1Main()
        shows VFr2Konv()
        shows VFr3Grohot()
        shows VFr7RandE()
        shows VFrADiag()
        shows VFr6Dedusting()
        shows VFr7RandE()
        shows VFrADiag()
    Button (633,95 100x70), "главная"
        OnMouseClick: FrameSelectionChange Selection=SelectedFrame=5ddc75d5-edde-4cc6-9f2a-3d195ac39671, GlobSel=AssignType=Directly, SelType=Locally
    Button (737,95 100x70), "конвейеры"
        OnMouseClick: FrameSelectionChange Selection=SelectedFrame=5ddc75d5-edde-4cc6-9f2a-3d195ac39671, Selection=1, GlobSel=AssignType=Directly, SelType=Locally
    Button (633,169 100x70), "3 конвейер грохот 2 конвейер"
        OnMouseClick: FrameSelectionChange Selection=SelectedFrame=5ddc75d5-edde-4cc6-9f2a-3d195ac39671, Selection=2, GlobSel=AssignType=Directly, SelType=Locally
    Button (737,169 100x70), input disabled if: TRUE
    Button (633,243 100x70), input disabled if: TRUE
    Button (737,243 100x70), input disabled if: TRUE
    Button (633,317 100x70), "готовности ошибки"
        OnMouseClick: FrameSelectionChange Selection=SelectedFrame=5ddc75d5-edde-4cc6-9f2a-3d195ac39671, Selection=3, GlobSel=AssignType=Directly, SelType=Locally
    Button (737,391 100x70), "Сброс"
        OnMouseDown: execute { PLC_PRG.xAck := TRUE; }
        OnMouseUp: execute { PLC_PRG.xAck := FALSE; }
    Button (737,317 100x70), input disabled if: TRUE
    Button (633,391 100x70), "диагно- стика"
        OnMouseClick: FrameSelectionChange Selection=SelectedFrame=5ddc75d5-edde-4cc6-9f2a-3d195ac39671, Selection=4, GlobSel=AssignType=Directly, SelType=Locally
    Rectangle (3,45 831x30), "Строка состояния", text list: 'STEPS', text index: Chain.Step
    Rectangle (545,4 288x30), "%t[dd.MM.yyyy HH:mm:ss]"
    Label (774,455 66x30), "21.12.24"
    Rectangle (354,7 150x30), "АВАРИЙНЫЙ СТОП", invisible if: PLC_PRG.DInput1.xDI1
    Rectangle (638,75 196x17), "Удаленное управление: %d", text variable: CountWebCli.iCountActivWebVisus, colour toggle: CountWebCli.xAlarm AND PLC_PRG.xFlash
    Image (4,3 145x40), image: ImagePool.333
    Label (722,455 75x30), "Дробь"
END_VISUALIZATION

// Device/Application/VFr1Main
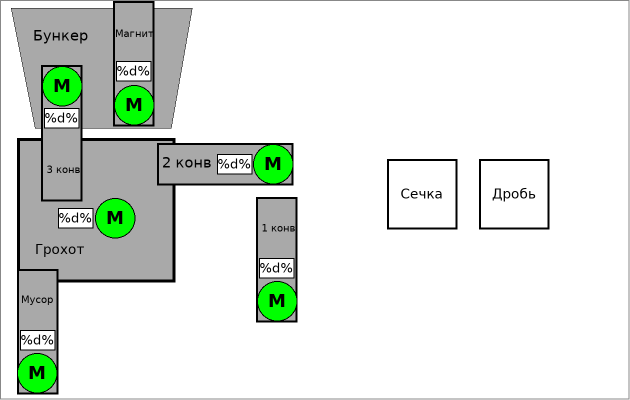
VISUALIZATION VFr1Main  // 630x400, background image ImagePool.fonFreame
    RoundedRectangle (17,138 158x144)
    Polygon (11,8) (85,8) (192,8) (171,128) (35,128)
    RoundedRectangle (256,197 41x125)
    RoundedRectangle (113,1 41x125)
    RoundedRectangle (17,269 41x125)
    RoundedRectangle (41,65 41x136)
    Ellipse (42,66 40x40), "М", colour toggle: MECH.K3.xOUT_Error
    Ellipse (17,353 40x40), "М", colour toggle: MECH.KMusor.xOUT_Error
    Ellipse (114,85 40x40), "М", colour toggle: MECH.KMagnit.xOUT_Error
    Ellipse (257,281 40x40), "М", colour toggle: MECH.K1.xOUT_Error
    Ellipse (95,198 40x40), "М", colour toggle: MECH.Gr.xOUT_Error
    Ellipse (42,66 40x40), "М", invisible if: NOT(MECH.K3.xOUT_Work)
    Ellipse (17,353 40x40), "М", invisible if: NOT(MECH.KMusor.xOUT_Work)
    Ellipse (114,85 40x40), "М", invisible if: NOT(MECH.KMagnit.xOUT_Work)
    Ellipse (257,281 40x40), "М", invisible if: NOT(MECH.K1.xOUT_Work)
    Ellipse (95,198 40x40), "М", invisible if: NOT(MECH.Gr.xOUT_Work)
    RoundedRectangle (157,143 136x42)
    Ellipse (253,144 40x40), "М", colour toggle: MECH.K2.xOUT_Error
    Ellipse (253,144 40x40), "М", invisible if: NOT(MECH.K2.xOUT_Work)
    RoundedRectangle (11,290 53x21), angle 270, "Мусор"
    RoundedRectangle (106,24 57x21), angle 270, "Магнит"
    RoundedRectangle (252,218 52x21), angle 270, "1 конв"
    RoundedRectangle (33,160 61x21), angle 270, "3 конв"
    RoundedRectangle (34,239 52x21), "Грохот"
    RoundedRectangle (24,16 73x39), "Бункер"
    RoundedRectangle (161,152 52x21), "2 конв"
    RoundedRectangle (20,330 35x20), "%d%", text variable: MECH.KMusor.iOUT_PVSpeed
    RoundedRectangle (116,61 35x20), "%d%", text variable: MECH.KMagnit.iOUT_PVSpeed
    RoundedRectangle (259,258 35x20), "%d%", text variable: MECH.KMagnit.iOUT_PVSpeed
    RoundedRectangle (58,208 35x20), "%d%", text variable: MECH.Gr.iOUT_PVSpeed
    RoundedRectangle (44,108 35x20), "%d%", text variable: MECH.K3.iOUT_PVSpeed
    RoundedRectangle (217,154 35x20), "%d%", text variable: MECH.K2.iOUT_PVSpeed
    RoundedRectangle (387,159 70x70), "Сечка", colour toggle: PLC_PRG.Sechka.Q1
    RoundedRectangle (479,159 70x70), "Дробь", colour toggle: PLC_PRG.Drob.Q1
END_VISUALIZATION

// Device/Application/VFr2Konv
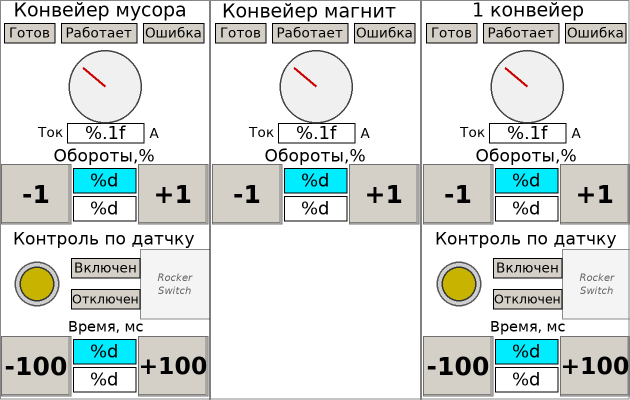
VISUALIZATION VFr2Konv  // 630x400, background image ImagePool.fonFreame
    Rectangle (73,196 63x25), "%d", text variable: MECH.KMusor.iOUT_PVSpeed
    Rectangle (73,168 63x25), "%d", text variable: MECH.KMusor_iIN_SPSpeed
    Button (138,164 70x60), "+1"
        OnMouseClick: execute {
            IF MECH.KMusor_iIN_SPSpeed <100 THEN
            	MECH.KMusor_iIN_SPSpeed := MECH.KMusor_iIN_SPSpeed + 1;
            END_IF;
        }
    Button (1,164 70x60), "-1"
        OnMouseClick: execute {
            IF MECH.KMusor_iIN_SPSpeed >5 THEN
            	MECH.KMusor_iIN_SPSpeed := MECH.KMusor_iIN_SPSpeed - 1;
            END_IF;
        }
    Label (15,0 170x20), "Конвейер мусора"
    Rectangle (67,123 77x20), "%.1f", text variable: MECH.KMusor.rOUT_Current
    Label (22,123 57x19), "Ток"
    Label (57,148 94x15), "Обороты,%"
    Rectangle (73,367 63x25), "%d", text variable: MECH.KMusor.iOUT_PVRotation, colour toggle: MECH.KonveerMusor.xFirstRun
    Rectangle (73,339 63x25), "%d", text variable: MECH.KMusor_iIN_SPRotatTimeMS
    Button (138,336 70x60), "+100"
        OnMouseClick: execute {
            IF MECH.KMusor_iIN_SPRotatTimeMS <10000 THEN
            	MECH.KMusor_iIN_SPRotatTimeMS := MECH.KMusor_iIN_SPRotatTimeMS + 100;
            END_IF;
        }
    Button (1,336 70x60), "-100"
        OnMouseClick: execute {
            IF MECH.KMusor_iIN_SPRotatTimeMS >500 THEN
            	MECH.KMusor_iIN_SPRotatTimeMS := MECH.KMusor_iIN_SPRotatTimeMS - 100;
            END_IF;
        }
    Label (2,229 204x19), "Контроль по датчку"
    RockerSwitch (140,249 70x70), variable: MECH.KMusor_xIN_EnCtrlSensor, behaviour: TOGGLE, style: Switch-RockerSwitch-Yellow
    Meter180 (33,50 144x73), value: MECH.KMusor.rOUT_Current, style: Meter-Meter180-Green, scale format: %d, scale 0..10
    Line (210,400) (210,0)
    Line (421,400) (421,0)
    Rectangle (61,23 76x20), "Работает", colour toggle: MECH.KMusor.xOUT_Work
    Rectangle (143,23 61x20), "Ошибка", colour toggle: MECH.KMusor.xOUT_Error
    Rectangle (4,23 51x20), "Готов", colour toggle: MECH.KMusor.xOUT_Ready
    Label (139,124 30x19), "А"
    Lamp1 (10,258 54x52), variable: PLC_PRG.DInput1.xDI15, style: Lamp-Lamp1-Yellow
    Label (4,317 204x19), "Время, мс"
    Rectangle (71,258 69x20), "Включен", colour toggle: MECH.KMusor_xIN_EnCtrlSensor
    Rectangle (71,289 69x20), "Отключен", colour toggle: NOT(MECH.KMusor_xIN_EnCtrlSensor)
    Rectangle (284,196 63x25), "%d", text variable: MECH.KMagnit.iOUT_PVSpeed
    Rectangle (284,168 63x25), "%d", text variable: MECH.KMagnit_iIN_SPSpeed
    Button (349,164 70x60), "+1"
        OnMouseClick: execute {
            IF MECH.KMagnit_iIN_SPSpeed <100 THEN
            	MECH.KMagnit_iIN_SPSpeed := MECH.KMagnit_iIN_SPSpeed + 1;
            END_IF;
        }
    Button (212,164 70x60), "-1"
        OnMouseClick: execute {
            IF MECH.KMagnit_iIN_SPSpeed >5 THEN
            	MECH.KMagnit_iIN_SPSpeed := MECH.KMagnit_iIN_SPSpeed - 1;
            END_IF;
        }
    Label (224,1 170x20), "Конвейер магнит"
    Rectangle (278,123 77x20), "%.1f", text variable: MECH.KMagnit.rOUT_Current
    Label (233,123 57x19), "Ток"
    Label (268,148 94x15), "Обороты,%"
    Meter180 (244,50 144x73), value: MECH.KMagnit.rOUT_Current, style: Meter-Meter180-Green, scale format: %d, scale 0..10
    Rectangle (272,23 76x20), "Работает", colour toggle: MECH.KMagnit.xOUT_Work
    Rectangle (354,23 61x20), "Ошибка", colour toggle: MECH.KMagnit.xOUT_Error
    Rectangle (215,23 51x20), "Готов", colour toggle: MECH.KMagnit.xOUT_Ready
    Label (350,124 30x19), "А"
    Rectangle (495,196 63x25), "%d", text variable: MECH.K1.iOUT_PVSpeed
    Rectangle (495,168 63x25), "%d", text variable: MECH.K1_iIN_SPSpeed
    Button (560,164 70x60), "+1"
        OnMouseClick: execute {
            IF MECH.K1_iIN_SPSpeed <100 THEN
            	MECH.K1_iIN_SPSpeed := MECH.K1_iIN_SPSpeed + 1;
            END_IF;
        }
    Button (423,164 70x60), "-1"
        OnMouseClick: execute {
            IF MECH.K1_iIN_SPSpeed >5 THEN
            	MECH.K1_iIN_SPSpeed := MECH.K1_iIN_SPSpeed - 1;
            END_IF;
        }
    Label (453,0 150x20), "1 конвейер"
    Rectangle (489,123 77x20), "%.1f", text variable: MECH.K1.rOUT_Current
    Label (444,123 57x19), "Ток"
    Label (479,148 94x15), "Обороты,%"
    Rectangle (495,367 63x25), "%d", text variable: MECH.K1.iOUT_PVRotation, colour toggle: MECH.Konveer1.xFirstRun
    Rectangle (495,339 63x25), "%d", text variable: MECH.K1_iIN_SPRotatTimeMS
    Button (560,336 70x60), "+100"
        OnMouseClick: execute {
            IF MECH.K1_iIN_SPRotatTimeMS <10000 THEN
            	MECH.K1_iIN_SPRotatTimeMS := MECH.K1_iIN_SPRotatTimeMS + 100;
            END_IF;
        }
    Button (423,336 70x60), "-100"
        OnMouseClick: execute {
            IF MECH.K1_iIN_SPRotatTimeMS >500 THEN
            	MECH.K1_iIN_SPRotatTimeMS := MECH.K1_iIN_SPRotatTimeMS - 100;
            END_IF;
        }
    RockerSwitch (562,249 70x70), variable: MECH.K1_xIN_EnCtrlSensor, behaviour: TOGGLE, style: Switch-RockerSwitch-Yellow
    Meter180 (455,50 144x73), value: MECH.K1.rOUT_Current, style: Meter-Meter180-Green, scale format: %d, scale 0..10
    Rectangle (483,23 76x20), "Работает", colour toggle: MECH.K1.xOUT_Work
    Rectangle (565,23 61x20), "Ошибка", colour toggle: MECH.K1.xOUT_Error
    Rectangle (426,23 51x20), "Готов", colour toggle: MECH.K1.xOUT_Ready
    Label (561,124 30x19), "А"
    Lamp1 (432,258 54x52), variable: PLC_PRG.DInput1.xDI17, style: Lamp-Lamp1-Yellow
    Rectangle (493,258 69x20), "Включен", colour toggle: MECH.K1_xIN_EnCtrlSensor
    Rectangle (493,289 69x20), "Отключен", colour toggle: NOT(MECH.K1_xIN_EnCtrlSensor)
    Label (214,230 204x19)
    Label (426,317 204x19), "Время, мс"
    Label (424,229 204x19), "Контроль по датчку"
END_VISUALIZATION

// Device/Application/VFr3Grohot
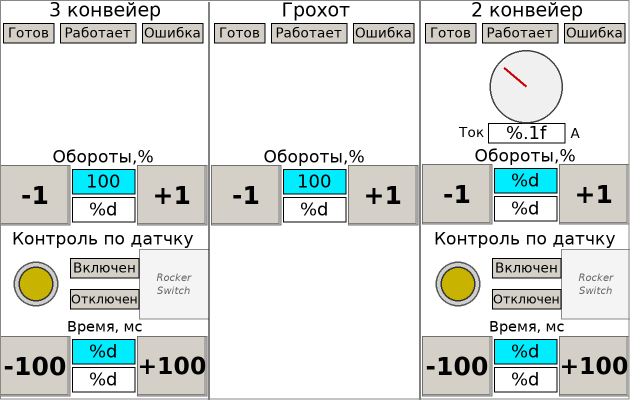
VISUALIZATION VFr3Grohot  // 630x400, background image ImagePool.fonFreame
    Label (40,0 130x20), "3 конвейер"
    Rectangle (72,367 63x25), "%d", text variable: MECH.K3.iOUT_PVRotation, colour toggle: MECH.Konveer3.xFirstRun
    Rectangle (72,339 63x25), "%d", text variable: MECH.K3_iIN_SPRotatTimeMS
    Button (137,336 70x60), "+100"
        OnMouseClick: execute {
            IF MECH.K3_iIN_SPRotatTimeMS <10000 THEN
            	MECH.K3_iIN_SPRotatTimeMS := MECH.K3_iIN_SPRotatTimeMS + 100;
            END_IF;
        }
    Label (1,229 204x19), "Контроль по датчку"
    RockerSwitch (139,249 70x70), variable: MECH.K3_xIN_EnCtrlSensor, behaviour: TOGGLE, style: Switch-RockerSwitch-Yellow
    Rectangle (60,23 76x20), "Работает", colour toggle: MECH.K3.xOUT_Work
    Rectangle (142,23 61x20), "Ошибка", colour toggle: MECH.K3.xOUT_Error
    Rectangle (3,23 51x20), "Готов", colour toggle: MECH.K3.xOUT_Ready
    Lamp1 (9,258 54x52), variable: PLC_PRG.DInput1.xDI18, style: Lamp-Lamp1-Yellow
    Label (3,317 204x19), "Время, мс"
    Rectangle (70,258 69x20), "Включен", colour toggle: MECH.K3_xIN_EnCtrlSensor
    Rectangle (70,289 69x20), "Отключен", colour toggle: NOT(MECH.K3_xIN_EnCtrlSensor)
    Label (251,0 130x20), "Грохот"
    Rectangle (271,23 76x20), "Работает", colour toggle: MECH.Gr.xOUT_Work
    Rectangle (353,23 61x20), "Ошибка", colour toggle: MECH.Gr.xOUT_Error
    Rectangle (214,23 51x20), "Готов", colour toggle: MECH.Gr.xOUT_Ready
    Rectangle (494,196 63x25), "%d", text variable: MECH.K2.iOUT_PVSpeed
    Rectangle (494,168 63x25), "%d", text variable: MECH.iSP_Konveer2
    Button (559,164 70x60), "+1", invisible if: TRUE
        OnMouseClick: execute {
            IF MECH.K2_iIN_SPSpeed <100 THEN
            	MECH.K2_iIN_SPSpeed := MECH.K2_iIN_SPSpeed + 1;
            END_IF;
        }
    Button (422,164 70x60), "-1", invisible if: TRUE
        OnMouseClick: execute {
            IF MECH.K2_iIN_SPSpeed >5 THEN
            	MECH.K2_iIN_SPSpeed := MECH.K2_iIN_SPSpeed - 1;
            END_IF;
        }
    Label (462,0 130x20), "2 конвейер"
    Rectangle (488,123 77x20), "%.1f", text variable: MECH.K2.rOUT_Current
    Label (443,123 57x19), "Ток"
    Label (478,148 94x15), "Обороты,%"
    Rectangle (494,367 63x25), "%d", text variable: MECH.K2.iOUT_PVRotation, colour toggle: MECH.Konveer2.xFirstRun
    Rectangle (494,339 63x25), "%d", text variable: MECH.K2_iIN_SPRotatTimeMS
    Button (559,336 70x60), "+100"
        OnMouseClick: execute {
            IF MECH.K2_iIN_SPRotatTimeMS <10000 THEN
            	MECH.K2_iIN_SPRotatTimeMS := MECH.K2_iIN_SPRotatTimeMS + 100;
            END_IF;
        }
    Button (422,336 70x60), "-100"
        OnMouseClick: execute {
            IF MECH.K2_iIN_SPRotatTimeMS >500 THEN
            	MECH.K2_iIN_SPRotatTimeMS := MECH.K2_iIN_SPRotatTimeMS - 100;
            END_IF;
        }
    RockerSwitch (561,249 70x70), variable: MECH.K2_xIN_EnCtrlSensor, behaviour: TOGGLE, style: Switch-RockerSwitch-Yellow
    Meter180 (454,50 144x73), value: MECH.K2.rOUT_Current, style: Meter-Meter180-Green, scale format: %d, scale 0..10
    Rectangle (482,23 76x20), "Работает", colour toggle: MECH.K2.xOUT_Work
    Rectangle (564,23 61x20), "Ошибка", colour toggle: MECH.K2.xOUT_Error
    Rectangle (425,23 51x20), "Готов", colour toggle: MECH.K2.xOUT_Ready
    Label (560,124 30x19), "А"
    Lamp1 (431,258 54x52), variable: PLC_PRG.DInput1.xDI19, style: Lamp-Lamp1-Yellow
    Rectangle (492,258 69x20), "Включен", colour toggle: MECH.K2_xIN_EnCtrlSensor
    Rectangle (492,289 69x20), "Отключен", colour toggle: NOT(MECH.K2_xIN_EnCtrlSensor)
    Label (425,317 204x19), "Время, мс"
    Label (423,229 204x19), "Контроль по датчку"
    Button (0,336 70x60), "-100"
        OnMouseClick: execute {
            IF MECH.K3_iIN_SPRotatTimeMS >500 THEN
            	MECH.K3_iIN_SPRotatTimeMS := MECH.K3_iIN_SPRotatTimeMS - 100;
            END_IF;
        }
    Line (209,402) (209,2)
    Line (420,400) (420,0)
    Button (211,165 70x60), "-1", input disabled if: TRUE
    Rectangle (283,197 63x25), "%d", text variable: MECH.Grohot.iOutPVSpeed
    Rectangle (283,169 63x25), "100"
    Button (348,165 70x60), "+1", input disabled if: TRUE
    Label (267,149 94x15), "Обороты,%"
    Button (0,165 70x60), "-1", input disabled if: TRUE
    Rectangle (72,197 63x25), "%d", text variable: MECH.Konveer3.iOutPVSpeed
    Rectangle (72,169 63x25), "100"
    Button (137,165 70x60), "+1", input disabled if: TRUE
    Label (56,149 94x15), "Обороты,%"
END_VISUALIZATION

// Device/Application/VFr7RandE
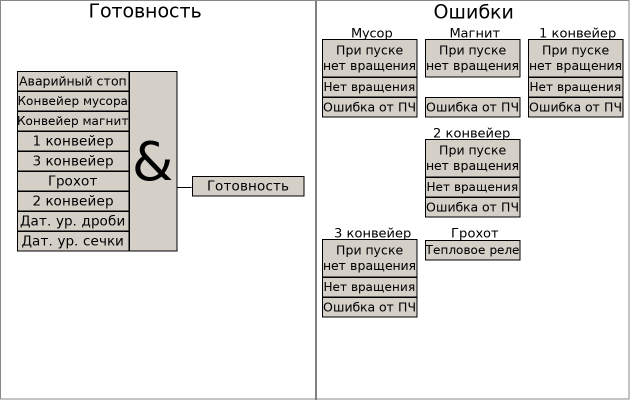
VISUALIZATION VFr7RandE  // 630x400, background image ImagePool.fonFreame
    Label (409,2 130x20), "Ошибки"
    Label (80,1 130x20), "Готовность"
    Line (316,401) (316,1)
    Rectangle (322,39 95x38), "При пуске нет вращения", colour toggle: MECH.KonveerMusor.xStartNoRotation
    Rectangle (17,71 112x20), "Аварийный стоп", colour toggle: PLC_PRG.DInput1.xDI1
    Rectangle (17,91 112x20), "Конвейер мусора", colour toggle: MECH.KMusor.xOUT_Ready
    Rectangle (17,111 112x20), "Конвейер магнит", colour toggle: MECH.KMagnit.xOUT_Ready
    Rectangle (17,131 112x20), "1 конвейер", colour toggle: MECH.K1.xOUT_Ready
    Rectangle (17,151 112x20), "3 конвейер", colour toggle: MECH.K3.xOUT_Ready
    Rectangle (17,171 112x20), "Грохот", colour toggle: MECH.Gr.xOUT_Ready
    Rectangle (17,191 112x20), "2 конвейер", colour toggle: MECH.K2.xOUT_Ready
    Rectangle (129,71 48x180), "&", colour toggle: Chain.ReadyRun
    Rectangle (192,176 112x20), "Готовность", colour toggle: Chain.ReadyRun
    Line (177,187) (191,187)
    Label (307,23 130x20), "Мусор"
    Rectangle (322,77 95x20), "Нет вращения", colour toggle: MECH.KonveerMusor.xNoRation
    Rectangle (322,97 95x20), "Ошибка от ПЧ", colour toggle: MECH.KonveerMusor.xExtError
    Rectangle (425,39 95x38), "При пуске нет вращения", colour toggle: MECH.KonveerMagnit.xStartNoRotation
    Label (410,23 130x20), "Магнит"
    Rectangle (425,97 95x20), "Ошибка от ПЧ", colour toggle: MECH.KonveerMagnit.xExtError
    Rectangle (528,39 95x38), "При пуске нет вращения", colour toggle: MECH.Konveer1.xStartNoRotation
    Label (513,23 130x20), "1 конвейер"
    Rectangle (528,77 95x20), "Нет вращения", colour toggle: MECH.Konveer1.xNoRation
    Rectangle (528,97 95x20), "Ошибка от ПЧ", colour toggle: MECH.Konveer1.xExtError
    Label (308,223 130x20), "3 конвейер"
    Rectangle (425,139 95x38), "При пуске нет вращения", colour toggle: MECH.Konveer2.xStartNoRotation
    Label (407,123 130x20), "2 конвейер"
    Rectangle (425,177 95x20), "Нет вращения", colour toggle: MECH.Konveer2.xNoRation
    Rectangle (425,197 95x20), "Ошибка от ПЧ", colour toggle: MECH.Konveer2.xExtError
    Rectangle (322,239 95x38), "При пуске нет вращения", colour toggle: MECH.Konveer3.xStartNoRotation
    Rectangle (322,277 95x20), "Нет вращения", colour toggle: MECH.Konveer3.xNoRation
    Label (410,223 130x20), "Грохот"
    Rectangle (425,240 95x20), "Тепловое реле", colour toggle: MECH.Grohot.xExtError
    Rectangle (322,297 95x20), "Ошибка от ПЧ", colour toggle: MECH.Konveer3.xExtError
    Rectangle (17,211 112x20), "Дат. ур. дроби", colour toggle: NOT(PLC_PRG.DInput1.xDI16)
    Rectangle (17,231 112x20), "Дат. ур. сечки", colour toggle: NOT(PLC_PRG.DInput1.xDI20)
END_VISUALIZATION

(* text list System (id | default)
  Apr | Apr
  April | April
  Aug | Aug
  August | August
  Dec | Dec
  December | December
  Feb | Feb
  February | February
  Fri | Fri
  Friday | Friday
  Jan | Jan
  January | January
  Jul | Jul
  July | July
  Jun | Jun
  June | June
  Mar | Mar
  March | March
  May | May
  May_3Letter | May
  Mon | Mon
  Monday | Monday
  Nov | Nov
  November | November
  Oct | Oct
  October | October
  Sat | Sat
  Saturday | Saturday
  Sep | Sep
  September | September
  Sun | Sun
  Sunday | Sunday
  Thu | Thu
  Thursday | Thursday
  Tue | Tue
  Tuesday | Tuesday
  Wed | Wed
  Wednesday | Wednesday
   |  *)
